// TwinCAT 3 PLC project TcLog_Sandboxx
// ProgramVersion: 3.1.4026.20
// libraries:
//   Tc2_Standard, * (Beckhoff Automation GmbH)
//   Tc2_System, * (Beckhoff Automation GmbH)
//   Tc2_Utilities, * (Beckhoff Automation GmbH)
//   Tc3_Module, * (Beckhoff Automation GmbH)
//   [TcLog], * (Benedikt Geisler)
// project tree:
//   Programs/ FileOpenMode.TcDUT, Main.TcPOU, RollingFileState.TcDUT, RollingFile.TcPOU
//   Tasks/ PlcTask.TcTTO
// real-time tasks:
//   TASK PlcTask: cycle T#10ms, priority 20, ADS port 350

CONFIGURATION TcLog_Sandboxx
    RESOURCE PLC ON TwinCAT3
        TASK PlcTask(INTERVAL := T#10ms, PRIORITY := 20);
        PROGRAM Main WITH PlcTask : Main;
    END_RESOURCE
END_CONFIGURATION

// ---- Programs/FileOpenMode.TcDUT
{attribute 'qualified_only'}
{attribute 'to_string'}
TYPE FileOpenMode :
(
	Read := Tc2_System.FOpen_ModeRead,
	Write := Tc2_System.FOpen_ModeWrite,
	Append := Tc2_System.FOpen_ModeAppend,
	Plus := Tc2_System.FOpen_ModePlus,
	Binary := Tc2_System.FOpen_ModeBinary,
	Text := Tc2_System.FOpen_ModeText
) DWORD;
END_TYPE

// ---- Programs/RollingFileState.TcDUT
{attribute 'qualified_only'}
{attribute 'strict'}
{attribute 'to_string'}
TYPE RollingFileState :
(
	Closed,
	Opening,
	Open,
	Closing,
	Writing,
	Error,
	RollingOver
);
END_TYPE

// ---- Programs/Main.TcPOU
PROGRAM Main
VAR
	f : RollingFile;	

	file_name : T_MaxString := 'C:\Logs\test.txt';
	open_file : BOOL;
	close_file : BOOL;
	line_to_write : T_MaxString := 'Gday cobber$L';
	write_line : BOOL;
	
	////////////////////////////////////////////////////////////////////////////////	

	core_logger : TcLogCore(BufferSize := 50 * 50 * (Tc2_System.MAX_STRING_LENGTH + Constants.FifoOverhead));
	logger : TcLog;
	ads_adapter : AdsLogTargetAdapter;
	file_adapter : FileLogTargetAdapter;
	
	trigger_log : BOOL;
	
	////////////////////////////////////////////////////////////////////////////////
	
	within_string : T_MaxString := 'this.is.a.test.log';
	found_index : INT;
	extension : T_MaxString;
	
	dev_id : DeviceIdentification;
	line : T_maxString;
END_VAR

IF open_file THEN
	f.Open(file_name, FileOpenMode.Append OR FileOpenMode.Text);
	
	IF f.IsOpen THEN
		open_file := FALSE;
	ELSIF f.IsErrored THEN
		open_file := FALSE;
	END_IF
END_IF

IF close_file THEN
	f.Close();
	
	IF f.IsClosed THEN
		close_file := FALSE;
	END_IF
END_IF

IF write_line THEN
	f.WriteString(line_to_write);
// 	IF  THEN
// 		write_line := FALSE;
// 	END_IF
END_IF

////////////////////////////////////////////////////////////////////////////////

found_index := FindLastOccurrence(within_string, '.');
extension := GetFileExtension(within_string);

dev_id.Initialise();

////////////////////////////////////////////////////////////////////////////////

core_logger
	.IncludeInstancePath()
	.MinimumLevel(LogLevel.Debug)
	.AddAdapter1(ads_adapter)
	.AddAdapter2(file_adapter
		.FilePath('C:\Users\User\workspaces\TcLog\logs')
		.FileName('tclog_sandbox.log')
		.SetRollingInterval(RollingInterval.Hourly)
		.DeleteLogFilesAfterDays(1))
	.RunLogger();

IF trigger_log THEN
	trigger_log := FALSE;
	logger.Debug('Yo');
END_IF

END_PROGRAM

// ---- Programs/RollingFile.TcPOU
FUNCTION_BLOCK RollingFile
VAR
	state : RollingFileState;
	file_open : Tc2_System.FB_FileOpen;
	file_close : Tc2_System.FB_FileClose;
	file_write : Tc2_System.FB_FileWrite;
	file_puts : Tc2_System.FB_FilePuts;
	file_handle : UINT;

	error_id : UDINT;

	lockFileWriteToForceRisingEdge : BOOL; // filePuts can only be executed every other cycle
									 // since it needs a rising edge to execute.
	net_id : T_AmsNetId := '';
END_VAR

METHOD PUBLIC Close : BOOL
VAR_INPUT
	timeout : TIME := Tc2_System.Default_Ads_Timeout;
END_VAR
IF state = RollingFileState.Open THEN
	file_close.hFile := file_handle;
	file_close.tTimeout := timeout;
	file_close.bExecute := TRUE;
	
	state := RollingFileState.Closing;
ELSIF state = RollingFileState.Closing THEN
	IF NOT file_close.bBusy THEN
		file_close.bExecute := FALSE;
		Close := TRUE;

		IF file_close.bError THEN
			error_id := file_close.nErrId;
			state := RollingFileState.Error;
		ELSE
			file_handle := 0;
			state := RollingFileState.Closed;
		END_IF
	END_IF	
END_IF

file_close();
END_METHOD

{attribute 'monitoring':='call'}
PROPERTY PUBLIC ErrorId : UDINT
GET // PUBLIC
ErrorId := error_id;
END_GET
END_PROPERTY

{attribute 'monitoring':='call'}
PROPERTY PUBLIC FileName : T_MaxString
GET // PUBLIC
FileName := SEL(IsOpen, '', file_open.sPathName);
END_GET
END_PROPERTY

{attribute 'monitoring':='call'}
PROPERTY PUBLIC IsClosed : BOOL
GET // PUBLIC
IsClosed := state = RollingFileState.Closed;
END_GET
END_PROPERTY

{attribute 'monitoring':='call'}
PROPERTY PUBLIC IsErrored : BOOL
GET // PUBLIC
IsErrored := state = RollingFileState.Error;
END_GET
END_PROPERTY

{attribute 'monitoring':='call'}
PROPERTY PUBLIC IsOpen : BOOL
GET // PUBLIC
IsOpen := state = RollingFileState.Open;
END_GET
END_PROPERTY

METHOD PUBLIC Open : BOOL
VAR_INPUT
	file_name : T_MaxString;
	mode : FileOpenMode;
	timeout : TIME := Tc2_System.Default_Ads_Timeout;
END_VAR
IF state = RollingFileState.Closed THEN
	file_open.sPathName := file_name;
	file_open.nMode := mode; 
	file_open.tTimeout := timeout;
	file_open.bExecute := TRUE;
	
	state := RollingFileState.Opening;
ELSIF state = RollingFileState.Opening THEN
	IF NOT file_open.bBusy THEN
		file_open.bExecute := FALSE;
		Open := TRUE;

		IF file_open.bError OR file_open.hFile = 0 THEN
			error_id := file_open.nErrId;
			state := RollingFileState.Error;
		ELSE
			file_handle := file_open.hFile;
			state := RollingFileState.Open;
		END_IF
	END_IF
END_IF

file_open(
	sNetId := net_id,
	ePath := Tc2_System.E_OpenPath.Path_Generic
);
END_METHOD

METHOD PUBLIC WriteString : BOOL
VAR_INPUT
	line : T_MaxString;
	timeout : TIME := Tc2_System.Default_Ads_Timeout;
END_VAR
IF state = RollingFileState.Open THEN
	file_puts.sLine := line;
	file_puts.tTimeout := timeout;
	file_puts.bExecute := TRUE;
	
	IF NOT file_puts.bBusy THEN
		file_puts.bExecute := FALSE;
		WriteString := TRUE;
		
		IF file_puts.bError THEN
			error_id := file_puts.nErrId;
			state := RollingFileState.Error;
		END_IF
	END_IF
END_IF

file_puts(
	sNetId := net_id,
	hFile := file_handle
);
END_METHOD

END_FUNCTION_BLOCK
